# EPICS substitutions: src/iocdoc/testfiles/iocBoot/ioc495idc/templates/xradia_motor.substitutions
file "$(TOP)/495idcApp/Db/xradia_motor.db"
{
pattern
{P          PORT  ADDR  N   M       DESC                   DIR  VBAS  VELO      VMAX     HVEL       ACCL   BDST  BVEL  BACC  MRES         PREC  EGU    DHLM        DLLM         HLM  LLM  RTRY  NTM    INIT}

{495idcnpi: pmac1  1     1  "m$(N)" "Objective X"          0    0      100.0    100.0     200.0     0.001  0     0     0     0.1          5     "um"       2000.0      -2000.0  0    0    0     "NO"   ""}
{495idcnpi: pmac1  2     2  "m$(N)" "Objective Z"          0    0      100.0    100.0     200.0     0.001  0     0     0     0.1          5     "um"       2000.0      -2000.0  0    0    0     "NO"   ""}
{495idcnpi: pmac1  3     3  "m$(N)" "Sample Chi (Tip)"     0    0        0.04     0.04      0.0133  0.001  0     0     0     0.000013333  5     "um"          2.0         -2.0  0    0    0     "NO"   ""}
{495idcnpi: pmac1  4     4  "m$(N)" "Sample Phi (Tilt)"    0    0        0.04     0.04      0.0133  0.001  0     0     0     0.000013333  5     "um"          2.0         -2.0  0    0    0     "NO"   ""}
{495idcnpi: pmac1  5     5  "m$(N)" "Condenser X"          0    0      200.0    200.0     200.0     0.001  0     0     0     0.1          5     "um"       2538.9     -39461.1  0    0    0     "NO"   ""}
{495idcnpi: pmac1  6     6  "m$(N)" "Condenser Y"          0    0      200.0    200.0     200.0     0.001  0     0     0     0.1          5     "um"       4441.9      -4000.0  0    0    0     "NO"   ""}
{495idcnpi: pmac1  7     7  "m$(N)" "Condenser Z"          0    0      200.0    200.0     200.0     0.001  0     0     0     0.1          5     "um"      10801.6      -9198.4  0    0    0     "NO"   ""}
{495idcnpi: pmac1  8     8  "m$(N)" "Condenser Tip"        0    0       31.75    31.75     38.1     0.001  0     0     0     0.0635       5     "um"       1000.0      -1000.0  0    0    0     "NO"   ""}
{495idcnpi: pmac1  9     9  "m$(N)" "Condenser Tilt"       0    0       31.75    31.75     38.1     0.001  0     0     0     0.0635       5     "um"       2000.0      -2000.0  0    0    0     "NO"   ""}
{495idcnpi: pmac1 10    10  "m$(N)" "Focus X"              0    0      200.0    200.0     200.0     0.001  0     0     0     0.1          5     "um"       4500.0      -4500.0  0    0    0     "NO"   ""}
{495idcnpi: pmac1 11    11  "m$(N)" "Focus Y"              0    0      200.0    200.0     200.0     0.001  0     0     0     0.1          5     "um"       4000.0      -4000.0  0    0    0     "NO"   ""}
{495idcnpi: pmac1 12    12  "m$(N)" "Focus Z"              0    0      200.0    200.0     200.0     0.001  0     0     0     0.1          5     "um"       2500.0      -3500.0  0    0    0     "NO"   ""}
{495idcnpi: pmac1 13    13  "m$(N)" "OSA X"                0    0       20.0     20.0      20.0     0.001  0     0     0     0.08         5     "um"       5300.8      -4699.2  0    0    0     "NO"   ""}
{495idcnpi: pmac1 14    14  "m$(N)" "OSA Y"                0    0       20.0     20.0      20.0     0.001  0     0     0     0.08         5     "um"       4889.2      -5110.8  0    0    0     "NO"   ""}
{495idcnpi: pmac1 15    15  "m$(N)" "OSA Z"                0    0       20.0     20.0      20.0     0.001  0     0     0     0.08         5     "um"       2032.0      -1888.0  0    0    0     "NO"   ""}
{495idcnpi: pmac1 16    16  "m$(N)" "Sample X"             0    0      200.0    200.0     200.0     0.001  0     0     0     0.1          5     "um"       4000.0      -4000.0  0    0    0     "NO"   ""}
{495idcnpi: pmac1 17    17  "m$(N)" "Sample Y"             0    0      200.0    200.0     200.0     0.001  0     0     0     0.1          5     "um"       4000.0      -4000.0  0    0    0     "NO"   ""}
{495idcnpi: pmac1 18    18  "m$(N)" "Sample Z"             0    0      200.0    200.0     200.0     0.001  0     0     0     0.1          5     "um"       1856.0      -2144.0  0    0    0     "NO"   ""}
{495idcnpi: pmac1 19    19  "m$(N)" "Metrology Rotation"   0    0        1.598    1.598     0.3196  0.001  0     0     0     0.0001598    5     "deg"         0.0          0.0  0    0    0     "NO"   ""}
{495idcnpi: pmac1 20    20  "m$(N)" "Sample Theta"         0    0        0.4      0.4       0.6     0.001  0     0     0     0.0002       5     "deg"        55.0        -55.0  0    0    0     "NO"   ""}
{495idcnpi: pmac1 21    21  "m$(N)" "Objective Y"          0    0      200.0    200.0     200.0     0.001  0     0     0     0.1          5     "um"       2200.0      -4005.0  0    0    0     "NO"   ""}
{495idcnpi: pmac1 22    22  "m$(N)" "Phase Ring X"         0    0       20.0     20.0      20.0     0.001  0     0     0     0.08         5     "um"       1600.0      -4800.0  0    0    0     "NO"   ""}
{495idcnpi: pmac1 23    23  "m$(N)" "Phase Ring Y"         0    0       20.0     20.0      20.0     0.001  0     0     0     0.08         5     "um"        800.0       -800.0  0    0    0     "NO"   ""}
{495idcnpi: pmac1 24    24  "m$(N)" "Phase Ring Z"         0    0       20.0     20.0      20.0     0.001  0     0     0     0.08         5     "um"       2000.0      -2000.0  0    0    0     "NO"   ""}
{495idcnpi: pmac1 25    25  "m$(N)" "Detector Low Z"       0    0     4000.0   4000.0    4000.0     0.001  0     0     0     1.0          5     "um"          0.0          0.0  0    0    0     "NO"   ""}
{495idcnpi: pmac1 26    26  "m$(N)" "Detector Mid Z"       0    0     4000.0   4000.0    4000.0     0.001  0     0     0     1.0          5     "um"          0.0          0.0  0    0    0     "NO"   ""}
{495idcnpi: pmac1 27    27  "m$(N)" "Detector Up Z"        0    0     4000.0   4000.0    4000.0     0.001  0     0     0     1.0          5     "um"          0.0          0.0  0    0    0     "NO"   ""}
{495idcnpi: pmac1 28    28  "m$(N)" "Intermediate Lens X"  0    0      195.3    195.3     195.3     0.001  0     0     0     0.009765     5     "um"        390.6      -4882.5  0    0    0     "NO"   ""}
{495idcnpi: pmac1 29    29  "m$(N)" "Tubelens"             0    0     1250.0   1250.0    2500.0     0.001  0     0     0     1.25         5     "um"   12500000.0  -12500000.0  0    0    0     "NO"   ""}

{495idcnpi: pmac2 34    34  "m$(N)" "ZP Piezo X"           0    0        3.75     3.75      4.0     0.001  0     0     0     0.000125     5     "um"          0.0          0.0  0    0    0     "NO"   ""}
{495idcnpi: pmac2 35    35  "m$(N)" "ZP Piezo Y"           0    0       10.0     10.0       4.0     0.001  0     0     0     0.000125     5     "um"          0.0          0.0  0    0    0     "NO"   ""}

}
